TYPE stErrorHandling :
STRUCT
	sTag: STRING;
	sMessage: STRING;
	sPriority: INT;
	sDevice: STRING;
	dErrorTime: DATE_AND_TIME;
	bIsAlarmAcknowledged : BOOL;
	bAcknowledged: BOOL;
	sPossibleSolution: STRING;
END_STRUCT
END_TYPE

(* stored: Version 1.1.0.1, ProductVersion 3.1.4024.12
   DUT stErrorHandling: Id {277228dd-be3d-4498-974f-425ac3d0325e} *)
